(* PLC project  *)

CONFIGURATION Empty_Module_23
END_CONFIGURATION
